TYPE NciPlc :
STRUCT
	nciToPlc AT %I* : NcToPlc_NciChannel_Ref;
	plcToNci AT %Q* : PlcToNc_NciChannel_Ref;
END_STRUCT
END_TYPE

(* stored: Version 1.1.0.1, ProductVersion 3.1.4024.12
   DUT NciPlc: Id {eecf8fdf-cee4-4994-8eaf-54a13a081492} *)
